// Mitsubishi GX Works2 project: 11. countter+sequence_3   PLC: Q03UDV

PROGRAM MAIN
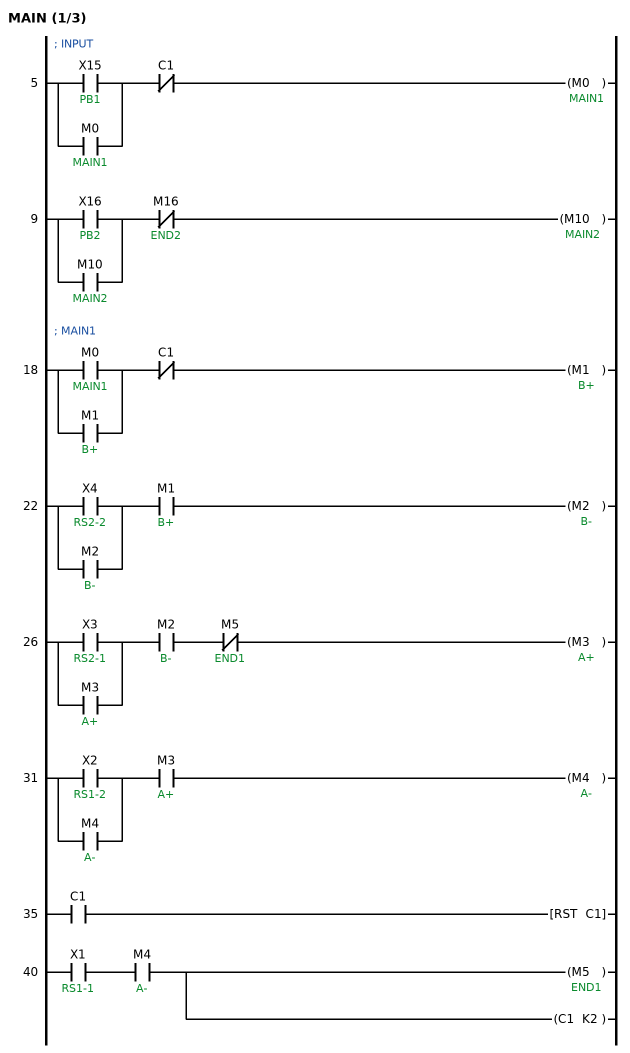
; INPUT
5     LD      X15  ; PB1
      OR      M0  ; MAIN1
      ANI     C1
      OUT     M0  ; MAIN1
9     LD      X16  ; PB2
      OR      M10  ; MAIN2
      ANI     M16  ; END2
      OUT     M10  ; MAIN2
; MAIN1
18    LD      M0  ; MAIN1
      OR      M1  ; B+
      ANI     C1
      OUT     M1  ; B+
22    LD      X4  ; RS2-2
      OR      M2  ; B-
      AND     M1  ; B+
      OUT     M2  ; B-
26    LD      X3  ; RS2-1
      OR      M3  ; A+
      AND     M2  ; B-
      ANI     M5  ; END1
      OUT     M3  ; A+
31    LD      X2  ; RS1-2
      OR      M4  ; A-
      AND     M3  ; A+
      OUT     M4  ; A-
35    LD      C1
      RST     C1
40    LD      X1  ; RS1-1
      AND     M4  ; A-
      OUT     M5  ; END1
      OUT     C1 K2
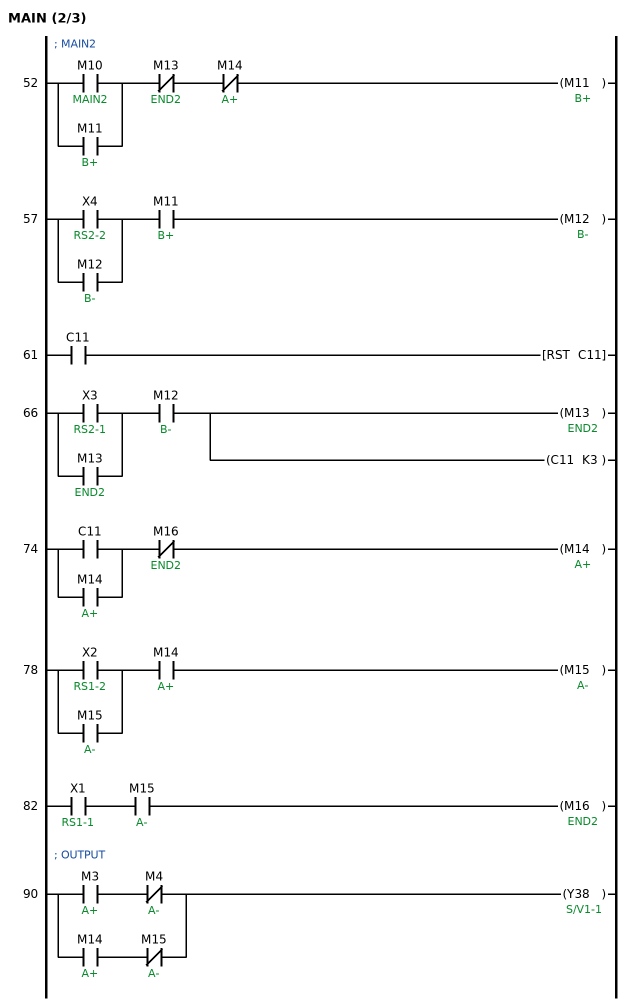
; MAIN2
52    LD      M10  ; MAIN2
      OR      M11  ; B+
      ANI     M13  ; END2
      ANI     M14  ; A+
      OUT     M11  ; B+
57    LD      X4  ; RS2-2
      OR      M12  ; B-
      AND     M11  ; B+
      OUT     M12  ; B-
61    LD      C11
      RST     C11
66    LD      X3  ; RS2-1
      OR      M13  ; END2
      AND     M12  ; B-
      OUT     M13  ; END2
      OUT     C11 K3
74    LD      C11
      OR      M14  ; A+
      ANI     M16  ; END2
      OUT     M14  ; A+
78    LD      X2  ; RS1-2
      OR      M15  ; A-
      AND     M14  ; A+
      OUT     M15  ; A-
82    LD      X1  ; RS1-1
      AND     M15  ; A-
      OUT     M16  ; END2
; OUTPUT
90    LD      M3  ; A+
      ANI     M4  ; A-
      LD      M14  ; A+
      ANI     M15  ; A-
      ORB
      OUT     Y38  ; S/V1-1
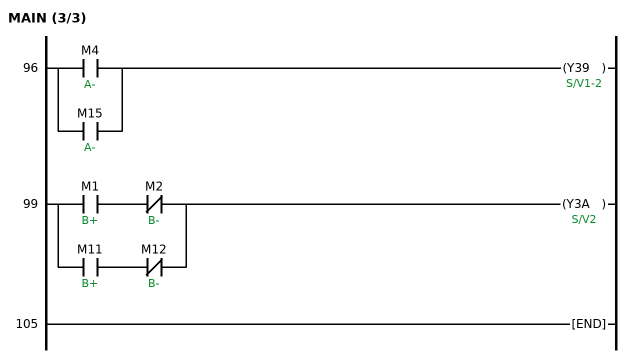
96    LD      M4  ; A-
      OR      M15  ; A-
      OUT     Y39  ; S/V1-2
99    LD      M1  ; B+
      ANI     M2  ; B-
      LD      M11  ; B+
      ANI     M12  ; B-
      ORB
      OUT     Y3A  ; S/V2
105   END
END_PROGRAM

// device comments not shown above
X17  ; PB3
X18  ; PB4
X1B  ; PB7
M20  ; MAIN3
M21  ; A+
M22  ; A-
M24  ; B+
M25  ; B-
M31  ; B+
M32  ; B-A+
M33  ; A-
